TYPE (* DataPanel Modules with medium IO density DO Struct + Source Address *)
  (* Version 1.0, 2026-05-28, franz *)
  PACKAGE DataPanel::io::MI::DQ;
  IMPORT DataPanel::io::MI::const::MI::MI_00;
  IMPORT DataPanel::io::MI::DQ::DataPanel_MI_DO_S;
  IMPORT DataPanel::io::MI::DQ::DataPanel_MI_DO::Invalid;
  DataPanel_MI_DO_S_Dual_SA : STRUCT
    u8SAMember : USINT := MI_00; (* Node SA 224..239 *)
    Up : DataPanel::io::MI::DQ::DataPanel_MI_DO_S := Invalid; (* Identify the Port 1A..8B forward, up, right, clockwise *)
    Down : DataPanel::io::MI::DQ::DataPanel_MI_DO_S := Invalid; (* Identify the Port 1A..8B backward, down, left, counter-clockwise *)
  END_STRUCT;
END_TYPE
